// TIA Portal project "tonrolesi_3adetmotor_kontrolu" (V18)

(* hardware
DEVICE "S7-1200 station_1"  S7-1200 Station
   slot 0: "Rack_0"  S7-1200 Rack  Rack  V1.0
   slot 1: "PLC_1"  CPU 1214C AC/DC/Rly  6ES7 214-1BG40-0XB0  V4.6
*)

// ===== PLC "PLC_1"  CPU 1214C AC/DC/Rly =====

VAR_GLOBAL   // PLC tag table "Default tag table"
   "STOP" AT %I0.0 : Bool;
   "START" AT %I0.1 : Bool;
   "Tag_1" AT %M0.0 : Bool;
   "Tag_2" AT %Q0.1 : Bool;
   "Tag_3" AT %Q0.2 : Bool;
   "Tag_4" AT %Q0.3 : Bool;
END_VAR

// folder: System blocks/Program resources

DATA_BLOCK "t1"   // DB1
{ S7_Optimized_Access := 'TRUE' }
AUTHOR : Simatic
FAMILY : IEC
NAME : IEC_TMR
VERSION : 1.0
// stored: InstanceOfName IEC_TIMER
"IEC_TIMER"
BEGIN
END_DATA_BLOCK

DATA_BLOCK "t2"   // DB2
{ S7_Optimized_Access := 'TRUE' }
AUTHOR : Simatic
FAMILY : IEC
NAME : IEC_TMR
VERSION : 1.0
// stored: InstanceOfName IEC_TIMER
"IEC_TIMER"
BEGIN
END_DATA_BLOCK

// folder: (top level)

ORGANIZATION_BLOCK "Main"   // OB1, LAD, ProgramCycle
TITLE = "Main Program Sweep (Cycle)"
{ S7_Optimized_Access := 'TRUE' }
VERSION : 0.1
   VAR_INPUT
      Initial_Call : Bool;   // Initial call of this OB
      Remanence : Bool;   // =True, if remanent data are available
   END_VAR
BEGIN

REGION Network 1
   // BİR SİSTEMDE 3 ADET MOTOR ÇALIŞACAKTIR. STARTA BASILDIĞINDA 1 VE 2.MOTOR ÇALIŞACAK. 10SN SONRA 1 DURACAK VE 3 ÇALIŞMAYA BAŞLAYACAK. 2 VE 3 BİRLİKTE 20SN ÇALIŞTIKTAN SONRA 2 DURACAK. 3 STOPA BASILANA KADARA ÇALIŞACAK
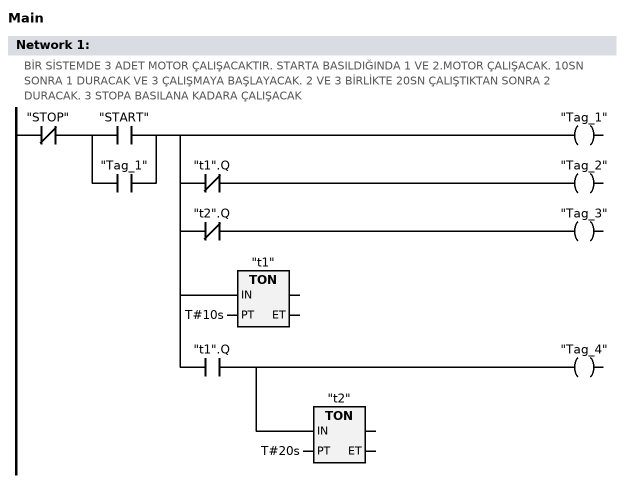
   "Tag_1" := NOT "STOP" AND ("START" OR "Tag_1");
   "Tag_2" := "Tag_1" AND NOT "t1".Q;
   "Tag_3" := "Tag_1" AND NOT "t2".Q;
   "t1".TON(IN := "Tag_1", PT := T#10s);
   "Tag_4" := "Tag_1" AND "t1".Q;
   "t2".TON(IN := "Tag_4", PT := T#20s);
END_REGION
END_ORGANIZATION_BLOCK